{attribute 'linkalways'} 
{attribute 'no_explicit_call' := 'This FB is a CLASS and must be accessed using methods or properties'}
{attribute 'enable_dynamic_creation'}
FUNCTION_BLOCK Node_F_VN_InvertMatrix3x3 EXTENDS VisionNode
VAR
    aSrcMatrix : _TcVnMatrix3x3_LREAL;
    aInvertedMatrix : _TcVnMatrix3x3_LREAL;
    hrPrev : _HRESULT(S_OK);
	hresult : _HRESULT(S_OK);
END_VAR

METHOD PUBLIC  Clone : I_Node
VAR
	pNode : POINTER TO Node_F_VN_InvertMatrix3x3;
END_VAR
pNode := __NEW(Node_F_VN_InvertMatrix3x3);
Clone := pNode^;
END_METHOD

METHOD FB_init : BOOL
VAR_INPUT
	bInitRetains : BOOL; // if TRUE, the retain variables are initialized (warm start / cold start)
	bInCopyCode : BOOL;  // if TRUE, the instance afterwards gets moved into the copy code (online change)
END_VAR
AddInput('aSrcMatrix', aSrcMatrix);
AddInput('hrPrev', hrPrev);
AddOutput('aInvertedMatrix', aInvertedMatrix);
AddOutput('hresult',hresult);
END_METHOD

METHOD PROTECTED OnExecute
hresult.Value := F_VN_InvertMatrix3x3(
	aSrcMatrix := aSrcMatrix.Value,
    aInvertedMatrix := aInvertedMatrix.Value,
	hrPrev:= hrPrev.Value);
END_METHOD

METHOD PUBLIC PreExecutionCheck
VAR_INPUT
	Check : I_PreExecutionChecks;
END_VAR
END_METHOD

END_FUNCTION_BLOCK

(* stored: Version 1.1.0.1, ProductVersion 3.1.4024.13
   POU Node_F_VN_InvertMatrix3x3: Id {3b20503a-8bfe-00b5-34f1-86f07118888b}, SpecialFunc None
   Folder Constructor: Id {7d1955ae-0539-0fdd-2866-599c93c6d838}
   Method Clone: Id {cf3a4313-fb4b-0911-1b9e-c2fc4589b72c}
   Method FB_init: Id {a401ac65-f89e-0951-1c00-67769feb26a7}
   Method OnExecute: Id {2b6dcc1f-ba06-0ffc-2cdf-81742ca1a655}
   Method PreExecutionCheck: Id {2f630c5f-5a63-0533-34a2-52d4ba38ac72} *)
